{attribute 'hide'}
{attribute clr [ExcludeFromApiDocumentation()]}
FUNCTION_BLOCK ABSTRACT _internals_TcoSequencer EXTENDS TcoSequencer

{attribute 'hide'}
METHOD PROTECTED FINAL _Close
THIS^.Close();
END_METHOD

{attribute 'hide'}
METHOD PROTECTED FINAL _Open
THIS^.Open();
END_METHOD

END_FUNCTION_BLOCK

(* stored: Version 1.1.0.1
   POU _internals_TcoSequencer: Id {8431c992-8d9f-09ad-1c50-56c92dc951c0}, SpecialFunc None
   Method _Close: Id {824aa06c-2eed-03ad-38e1-2b6360af64a5}
   Method _Open: Id {b37d3c58-1c1c-0875-2c6f-fc22d4441f2e} *)
